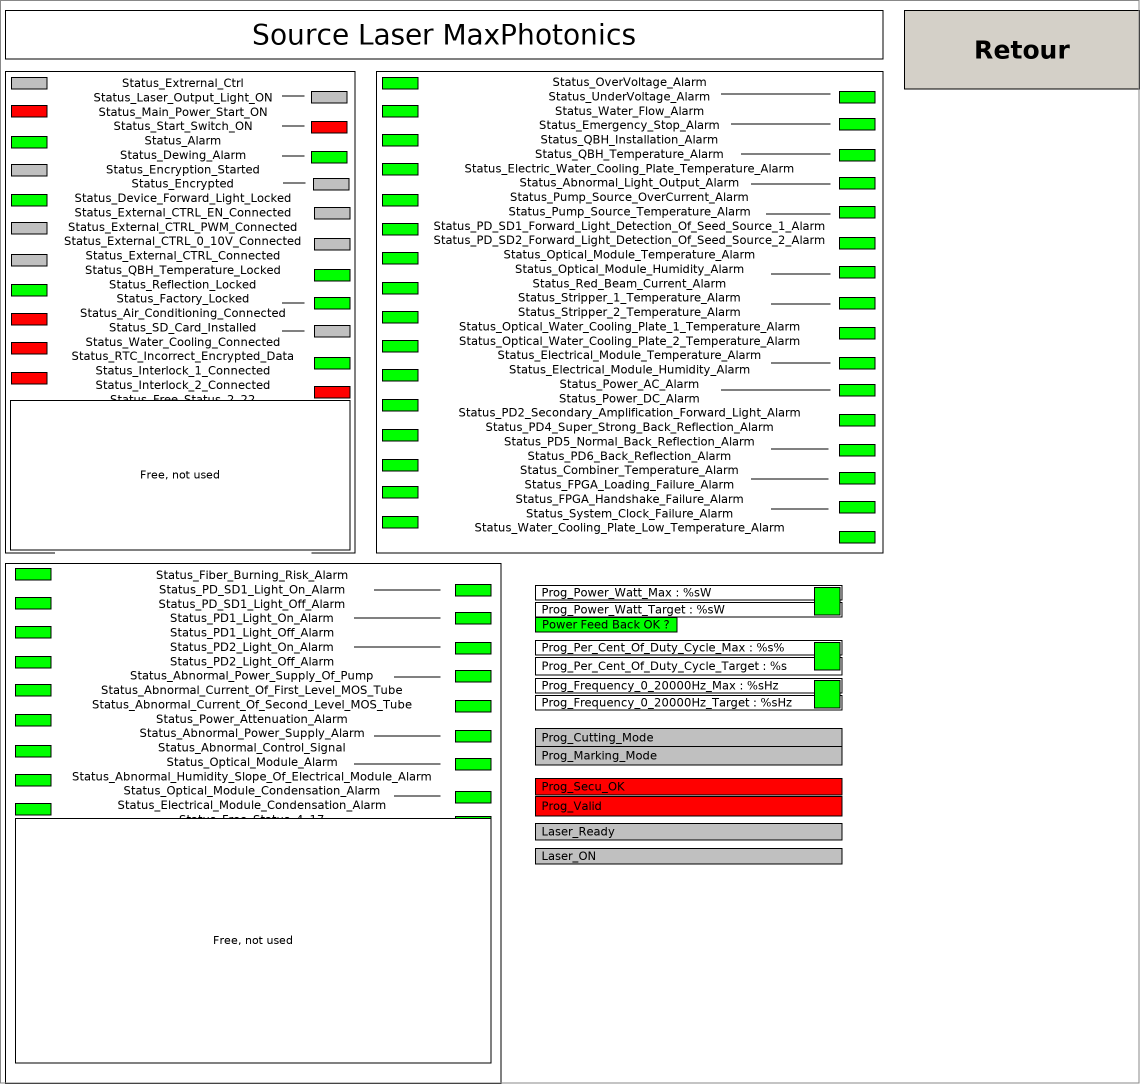
VISUALIZATION Visualization_source  // 1140x1084
    Rectangle (5,563 496x521)
    Rectangle (376,71 507x482)
    Rectangle (5,71 350x482)
    Rectangle (55,75 256x478), "Status_Extrernal_Ctrl Status_Laser_Output_Light_ON Status_Main_Power_Start_ON Status_Start_Switch_ON Status_Alarm Status_Dewing_Alarm Status_Encryption_Started Status_Encrypted Status_Device_Forward_Light_Locked Status_External_CTRL_EN_Connected Status_External_CTRL_PWM_Connected Status_External_CTRL_0_10V_Connected Status_External_CTRL_Connected Status_QBH_Temperature_Locked Status_Reflection_Locked Status_Factory_Locked Status_Air_Conditioning_Connected Status_SD_Card_Installed Status_Water_Cooling_Connected Status_RTC_Incorrect_Encrypted_Data Status_Interlock_1_Connected Status_Interlock_2_Connected Status_Free_Status_2_22 Status_Free_Status_2_23 Status_Free_Status_2_24 Status_Free_Status_2_25 Status_Free_Status_2_26 Status_Free_Status_2_27 Status_Free_Status_2_28 Status_Free_Status_2_29 Status_Free_Status_2_30 Status_Free_Status_2_31"
    Rectangle (424,74 411x477), "Status_OverVoltage_Alarm Status_UnderVoltage_Alarm Status_Water_Flow_Alarm Status_Emergency_Stop_Alarm Status_QBH_Installation_Alarm Status_QBH_Temperature_Alarm Status_Electric_Water_Cooling_Plate_Temperature_Alarm Status_Abnormal_Light_Output_Alarm Status_Pump_Source_OverCurrent_Alarm Status_Pump_Source_Temperature_Alarm Status_PD_SD1_Forward_Light_Detection_Of_Seed_Source_1_Alarm Status_PD_SD2_Forward_Light_Detection_Of_Seed_Source_2_Alarm Status_Optical_Module_Temperature_Alarm Status_Optical_Module_Humidity_Alarm Status_Red_Beam_Current_Alarm Status_Stripper_1_Temperature_Alarm Status_Stripper_2_Temperature_Alarm Status_Optical_Water_Cooling_Plate_1_Temperature_Alarm Status_Optical_Water_Cooling_Plate_2_Temperature_Alarm Status_Electrical_Module_Temperature_Alarm Status_Electrical_Module_Humidity_Alarm Status_Power_AC_Alarm Status_Power_DC_Alarm Status_PD2_Secondary_Amplification_Forward_Light_Alarm Status_PD4_Super_Strong_Back_Reflection_Alarm Status_PD5_Normal_Back_Reflection_Alarm Status_PD6_Back_Reflection_Alarm Status_Combiner_Temperature_Alarm Status_FPGA_Loading_Failure_Alarm Status_FPGA_Handshake_Failure_Alarm Status_System_Clock_Failure_Alarm Status_Water_Cooling_Plate_Low_Temperature_Alarm"
    Rectangle (11,77 36x12), colour toggle: SOURCE_MAXPHOTONICS.STATUS_2.0
    Rectangle (311,91 36x12), colour toggle: SOURCE_MAXPHOTONICS.STATUS_2.1
    Rectangle (11,105 36x12), colour toggle: SOURCE_MAXPHOTONICS.STATUS_2.2
    Rectangle (311,121 36x12), colour toggle: SOURCE_MAXPHOTONICS.STATUS_2.3
    Rectangle (382,77 36x12), colour toggle: SOURCE_MAXPHOTONICS.STATUS_3.0
    Rectangle (839,91 36x12), colour toggle: SOURCE_MAXPHOTONICS.STATUS_3.1
    Rectangle (382,105 36x12), colour toggle: SOURCE_MAXPHOTONICS.STATUS_3.2
    Rectangle (839,118 36x12), colour toggle: SOURCE_MAXPHOTONICS.STATUS_3.3
    Rectangle (382,134 36x12), colour toggle: SOURCE_MAXPHOTONICS.STATUS_3.4
    Rectangle (839,149 36x12), colour toggle: SOURCE_MAXPHOTONICS.STATUS_3.5
    Rectangle (382,163 36x12), colour toggle: SOURCE_MAXPHOTONICS.STATUS_3.6
    Rectangle (839,177 36x12), colour toggle: SOURCE_MAXPHOTONICS.STATUS_3.7
    Rectangle (382,194 36x12), colour toggle: SOURCE_MAXPHOTONICS.STATUS_3.8
    Rectangle (839,206 36x12), colour toggle: SOURCE_MAXPHOTONICS.STATUS_3.9
    Rectangle (382,223 36x12), colour toggle: SOURCE_MAXPHOTONICS.STATUS_3.10
    Rectangle (839,237 36x12), colour toggle: SOURCE_MAXPHOTONICS.STATUS_3.11
    Rectangle (382,252 36x12), colour toggle: SOURCE_MAXPHOTONICS.STATUS_3.12
    Rectangle (839,266 36x12), colour toggle: SOURCE_MAXPHOTONICS.STATUS_3.13
    Rectangle (382,282 36x12), colour toggle: SOURCE_MAXPHOTONICS.STATUS_3.14
    Rectangle (839,297 36x12), colour toggle: SOURCE_MAXPHOTONICS.STATUS_3.15
    Rectangle (382,311 36x12), colour toggle: SOURCE_MAXPHOTONICS.STATUS_3.16
    Rectangle (839,327 36x12), colour toggle: SOURCE_MAXPHOTONICS.STATUS_3.17
    Rectangle (382,340 36x12), colour toggle: SOURCE_MAXPHOTONICS.STATUS_3.18
    Rectangle (839,357 36x12), colour toggle: SOURCE_MAXPHOTONICS.STATUS_3.19
    Rectangle (382,369 36x12), colour toggle: SOURCE_MAXPHOTONICS.STATUS_3.20
    Rectangle (839,384 36x12), colour toggle: SOURCE_MAXPHOTONICS.STATUS_3.21
    Rectangle (382,399 36x12), colour toggle: SOURCE_MAXPHOTONICS.STATUS_3.22
    Rectangle (839,414 36x12), colour toggle: SOURCE_MAXPHOTONICS.STATUS_3.23
    Rectangle (382,429 36x12), colour toggle: SOURCE_MAXPHOTONICS.STATUS_3.24
    Rectangle (839,444 36x12), colour toggle: SOURCE_MAXPHOTONICS.STATUS_3.25
    Rectangle (382,459 36x12), colour toggle: SOURCE_MAXPHOTONICS.STATUS_3.26
    Rectangle (839,472 36x12), colour toggle: SOURCE_MAXPHOTONICS.STATUS_3.27
    Rectangle (382,486 36x12), colour toggle: SOURCE_MAXPHOTONICS.STATUS_3.28
    Rectangle (839,501 36x12), colour toggle: SOURCE_MAXPHOTONICS.STATUS_3.29
    Rectangle (382,516 36x12), colour toggle: SOURCE_MAXPHOTONICS.STATUS_3.30
    Rectangle (839,531 36x12), colour toggle: SOURCE_MAXPHOTONICS.STATUS_3.31
    Rectangle (11,136 36x12), colour toggle: SOURCE_MAXPHOTONICS.STATUS_2.4
    Rectangle (311,151 36x12), colour toggle: SOURCE_MAXPHOTONICS.STATUS_2.5
    Rectangle (11,164 36x12), colour toggle: SOURCE_MAXPHOTONICS.STATUS_2.6
    Rectangle (313,178 36x12), colour toggle: SOURCE_MAXPHOTONICS.STATUS_2.7
    Rectangle (11,194 36x12), colour toggle: SOURCE_MAXPHOTONICS.STATUS_2.8
    Rectangle (314,207 36x12), colour toggle: SOURCE_MAXPHOTONICS.STATUS_2.9
    Rectangle (11,222 36x12), colour toggle: SOURCE_MAXPHOTONICS.STATUS_2.10
    Rectangle (314,238 36x12), colour toggle: SOURCE_MAXPHOTONICS.STATUS_2.11
    Rectangle (11,254 36x12), colour toggle: SOURCE_MAXPHOTONICS.STATUS_2.12
    Rectangle (314,269 36x12), colour toggle: SOURCE_MAXPHOTONICS.STATUS_2.13
    Rectangle (11,284 36x12), colour toggle: SOURCE_MAXPHOTONICS.STATUS_2.14
    Rectangle (314,297 36x12), colour toggle: SOURCE_MAXPHOTONICS.STATUS_2.15
    Rectangle (11,313 36x12), colour toggle: SOURCE_MAXPHOTONICS.STATUS_2.16
    Rectangle (314,325 36x12), colour toggle: SOURCE_MAXPHOTONICS.STATUS_2.17
    Rectangle (11,342 36x12), colour toggle: SOURCE_MAXPHOTONICS.STATUS_2.18
    Rectangle (314,357 36x12), colour toggle: SOURCE_MAXPHOTONICS.STATUS_2.19
    Rectangle (11,372 36x12), colour toggle: SOURCE_MAXPHOTONICS.STATUS_2.20
    Rectangle (314,386 36x12), colour toggle: SOURCE_MAXPHOTONICS.STATUS_2.21
    Rectangle (11,400 36x12), colour toggle: SOURCE_MAXPHOTONICS.STATUS_2.22
    Rectangle (314,413 36x12), colour toggle: SOURCE_MAXPHOTONICS.STATUS_2.23
    Rectangle (11,430 36x12), colour toggle: SOURCE_MAXPHOTONICS.STATUS_2.24
    Rectangle (314,443 36x12), colour toggle: SOURCE_MAXPHOTONICS.STATUS_2.25
    Rectangle (11,459 36x12), colour toggle: SOURCE_MAXPHOTONICS.STATUS_2.26
    Rectangle (314,472 36x12), colour toggle: SOURCE_MAXPHOTONICS.STATUS_2.27
    Rectangle (11,487 36x12), colour toggle: SOURCE_MAXPHOTONICS.STATUS_2.28
    Rectangle (314,502 36x12), colour toggle: SOURCE_MAXPHOTONICS.STATUS_2.29
    Rectangle (11,517 36x12), colour toggle: SOURCE_MAXPHOTONICS.STATUS_2.30
    Rectangle (314,534 36x12), colour toggle: SOURCE_MAXPHOTONICS.STATUS_2.31
    Rectangle (52,567 400x514), "Status_Fiber_Burning_Risk_Alarm Status_PD_SD1_Light_On_Alarm Status_PD_SD1_Light_Off_Alarm Status_PD1_Light_On_Alarm Status_PD1_Light_Off_Alarm Status_PD2_Light_On_Alarm Status_PD2_Light_Off_Alarm Status_Abnormal_Power_Supply_Of_Pump Status_Abnormal_Current_Of_First_Level_MOS_Tube Status_Abnormal_Current_Of_Second_Level_MOS_Tube Status_Power_Attenuation_Alarm Status_Abnormal_Power_Supply_Alarm Status_Abnormal_Control_Signal Status_Optical_Module_Alarm Status_Abnormal_Humidity_Slope_Of_Electrical_Module_Alarm Status_Optical_Module_Condensation_Alarm Status_Electrical_Module_Condensation_Alarm Status_Free_Status_4_17 Status_Free_Status_4_18 Status_Free_Status_4_19 Status_Free_Status_4_20 Status_Free_Status_4_21 Status_Free_Status_4_22 Status_Free_Status_4_23 Status_Free_Status_4_24 Status_Free_Status_4_25 Status_Free_Status_4_26 Status_Free_Status_4_27 Status_Free_Status_4_28 Status_Free_Status_4_29 Status_Free_Status_4_30 Status_Free_Status_4_31"
    Rectangle (15,568 36x12), colour toggle: SOURCE_MAXPHOTONICS.STATUS_4.0
    Rectangle (455,584 36x12), colour toggle: SOURCE_MAXPHOTONICS.STATUS_4.1
    Rectangle (15,597 36x12), colour toggle: SOURCE_MAXPHOTONICS.STATUS_4.2
    Rectangle (455,612 36x12), colour toggle: SOURCE_MAXPHOTONICS.STATUS_4.3
    Rectangle (15,626 36x12), colour toggle: SOURCE_MAXPHOTONICS.STATUS_4.4
    Rectangle (455,642 36x12), colour toggle: SOURCE_MAXPHOTONICS.STATUS_4.5
    Rectangle (15,656 36x12), colour toggle: SOURCE_MAXPHOTONICS.STATUS_4.6
    Rectangle (455,670 36x12), colour toggle: SOURCE_MAXPHOTONICS.STATUS_4.7
    Rectangle (15,684 36x12), colour toggle: SOURCE_MAXPHOTONICS.STATUS_4.8
    Rectangle (455,700 36x12), colour toggle: SOURCE_MAXPHOTONICS.STATUS_4.9
    Rectangle (15,714 36x12), colour toggle: SOURCE_MAXPHOTONICS.STATUS_4.10
    Rectangle (455,730 36x12), colour toggle: SOURCE_MAXPHOTONICS.STATUS_4.11
    Rectangle (15,745 36x12), colour toggle: SOURCE_MAXPHOTONICS.STATUS_4.12
    Rectangle (455,758 36x12), colour toggle: SOURCE_MAXPHOTONICS.STATUS_4.13
    Rectangle (15,774 36x12), colour toggle: SOURCE_MAXPHOTONICS.STATUS_4.14
    Rectangle (455,791 36x12), colour toggle: SOURCE_MAXPHOTONICS.STATUS_4.15
    Rectangle (15,803 36x12), colour toggle: SOURCE_MAXPHOTONICS.STATUS_4.16
    Rectangle (455,816 36x12), colour toggle: SOURCE_MAXPHOTONICS.STATUS_4.17
    Rectangle (15,832 36x12), colour toggle: SOURCE_MAXPHOTONICS.STATUS_4.18
    Rectangle (455,848 36x12), colour toggle: SOURCE_MAXPHOTONICS.STATUS_4.19
    Rectangle (15,861 36x12), colour toggle: SOURCE_MAXPHOTONICS.STATUS_4.20
    Rectangle (455,878 36x12), colour toggle: SOURCE_MAXPHOTONICS.STATUS_4.21
    Rectangle (15,889 36x12), colour toggle: SOURCE_MAXPHOTONICS.STATUS_4.22
    Rectangle (455,904 36x12), colour toggle: SOURCE_MAXPHOTONICS.STATUS_4.23
    Rectangle (15,918 36x12), colour toggle: SOURCE_MAXPHOTONICS.STATUS_4.24
    Rectangle (455,936 36x12), colour toggle: SOURCE_MAXPHOTONICS.STATUS_4.25
    Rectangle (15,948 36x12), colour toggle: SOURCE_MAXPHOTONICS.STATUS_4.26
    Rectangle (455,966 36x12), colour toggle: SOURCE_MAXPHOTONICS.STATUS_4.27
    Rectangle (15,978 36x12), colour toggle: SOURCE_MAXPHOTONICS.STATUS_4.28
    Rectangle (455,995 36x12), colour toggle: SOURCE_MAXPHOTONICS.STATUS_4.29
    Rectangle (15,1008 36x12), colour toggle: SOURCE_MAXPHOTONICS.STATUS_4.30
    Rectangle (455,1024 36x12), colour toggle: SOURCE_MAXPHOTONICS.STATUS_4.31
    Rectangle (5,10 878x49), "Source Laser MaxPhotonics"
    Rectangle (535,585 307x15), "Prog_Power_Watt_Max : %sW", text variable: PLC_Prog_Power_Watt_Max
    Rectangle (535,602 307x15), "Prog_Power_Watt_Target : %sW", text variable: PLC_Prog_Power_Watt_Target
    Rectangle (535,640 307x15), "Prog_Per_Cent_Of_Duty_Cycle_Max : %s%", text variable: PLC_Prog_Per_Cent_Of_Duty_Cycle_Max
    Rectangle (535,657 307x18), "Prog_Per_Cent_Of_Duty_Cycle_Target : %s", text variable: PLC_Prog_Per_Cent_Of_Duty_Cycle_Target
    Rectangle (535,678 307x15), "Prog_Frequency_0_20000Hz_Max : %sHz", text variable: PLC_Prog_Frequency_0_20000Hz_Max
    Rectangle (535,695 307x15), "Prog_Frequency_0_20000Hz_Target : %sHz", text variable: PLC_Prog_Frequency_0_20000Hz_Target
    Rectangle (535,728 307x19), "Prog_Cutting_Mode", colour toggle: Prog_Cutting_Mode
    Rectangle (535,746 307x19), "Prog_Marking_Mode", colour toggle: Prog_Marking_Mode
    Rectangle (535,778 307x17), "Prog_Secu_OK", colour toggle: Prog_Secu_Source_OK
    Rectangle (814,587 26x28), colour toggle: Prog_Defaut_power_Watt_Target
    Rectangle (814,642 26x28), colour toggle: Prog_Defaut_Per_Cent_Of_Duty_Cycle_Target
    Rectangle (814,680 26x28), colour toggle: Prog_Defaut_Laser_Frequency_Of_PWM_Wave_Target
    Rectangle (535,617 142x15), "Power Feed Back OK ?", colour toggle: Prog_Defaut_Perc_Cent_Of_Laser_Output_Power_FeedBack
    Rectangle (535,848 307x16), "Laser_ON", colour toggle: SOURCE_MAXPHOTONICS.STATUS_2.1
    Rectangle (535,823 307x17), "Laser_Ready", colour toggle: SOURCE_MAXPHOTONICS.STATUS_2.1
    Rectangle (904,10 236x79), "Retour"
        OnMouseClick: change screen: MenuPrincipal
    Rectangle (535,796 307x20), "Prog_Valid", colour toggle: _1_LASER.FB_LASER_SOURCE_MAXPHOTONICS1.Prog_Valid
    Line (304,96) (282,96)
    Line (304,126) (282,126)
    Line (304,156) (282,156)
    Line (305,183) (283,183)
    Line (304,303) (282,303)
    Line (304,331) (282,331)
    Line (304,419) (282,419)
    Line (304,449) (282,449)
    Line (304,509) (282,509)
    Line (304,479) (282,479)
    Line (304,539) (282,539)
    Line (830,94) (721,94)
    Line (830,124) (731,124)
    Line (830,184) (751,184)
    Line (830,154) (741,154)
    Line (830,214) (766,214)
    Line (830,274) (771,274)
    Line (830,304) (771,304)
    Line (830,363) (771,363)
    Line (830,390) (721,390)
    Line (828,449) (771,449)
    Line (828,509) (771,509)
    Line (828,479) (751,479)
    Line (440,590) (374,590)
    Line (440,618) (354,618)
    Line (440,647) (354,647)
    Line (440,677) (394,677)
    Line (440,736) (374,736)
    Line (440,764) (354,764)
    Line (440,796) (394,796)
    Line (440,823) (344,823)
    Line (440,853) (344,853)
    Line (440,880) (344,880)
    Line (440,910) (344,910)
    Line (439,942) (343,942)
    Line (439,972) (343,972)
    Line (439,999) (343,999)
    Line (439,1029) (343,1029)
    Line (160,839) (64,839)
    Line (160,868) (64,868)
    Line (160,895) (64,895)
    Line (160,925) (64,925)
    Line (159,957) (63,957)
    Line (159,987) (63,987)
    Line (159,1014) (63,1014)
    Rectangle (15,818 476x245), "Free, not used"
    Rectangle (10,400 340x150), "Free, not used"
END_VISUALIZATION

(* stored: Version 1.1.0.1
   Visu Visualization_source: Id {36def81b-6339-4459-b273-f93866a865b9} *)
